(* Logix 5000 project; controller ecust2024 vendor 1 type 14 code 108 rev 30.11; software revision 30.00; part 2 of 2 *)
(* tags used below, declared in another part *)
   circle_count : DINT;
   circle_num1 : DINT;
   count11 : COUNTER;
   delay4 : TIMER;
   LED1 : LED_control;
   LED2 : LED_control;
   LED3 : LED_control;
   speed_dec : BOOL;
   speed_inc : BOOL;
   velocity : DINT;
   wait1 : TIMER;
   wait2 : TIMER;
   wait3 : TIMER;
   A : OneKey;
   anticlockwise : MOTION_INSTRUCTION;
   anticlockwise_order : BOOL;
   Axis_1 : AXIS_CIP_DRIVE;
   Change_speed : BOOL;
   changespeed : MOTION_INSTRUCTION;
   clockwise1 : MOTION_INSTRUCTION;
   clockwise_order : BOOL;
   count5 : COUNTER;
   count6 : COUNTER;
   Direction_Change3 : BOOL;
   Direction_Change4 : BOOL;
   Direction_change_state3 : BOOL;
   Holding_Cmd : BOOL;
   Light1 : BOOL;
   Light2 : BOOL;
   Light3 : BOOL;
   LT1 : BOOL;
   LT2 : BOOL;
   LT3 : BOOL;
   My_Equipment_Phase : PHASE;
   oneshot : DINT;
   Reset_Cmd : BOOL;
   Restart_Cmd : BOOL;
   S : DINT;
   Sensor1_cmd : BOOL;
   Sensor2_cmd : BOOL;
   setspeed : DINT;
   Start_Cmd : BOOL;
   Start_PB : BOOL;
   StartA : BOOL;
   Stop : MOTION_INSTRUCTION;
   Stop_Cmd : BOOL;
   Stop_PB : BOOL;
   Temp_CMX : REAL;
   temperature_speed : REAL;
   time1 : TIMER;
   time2 : TIMER;
   time4 : TIMER;
   ts : BOOL;
(* MainProgram, continued *)

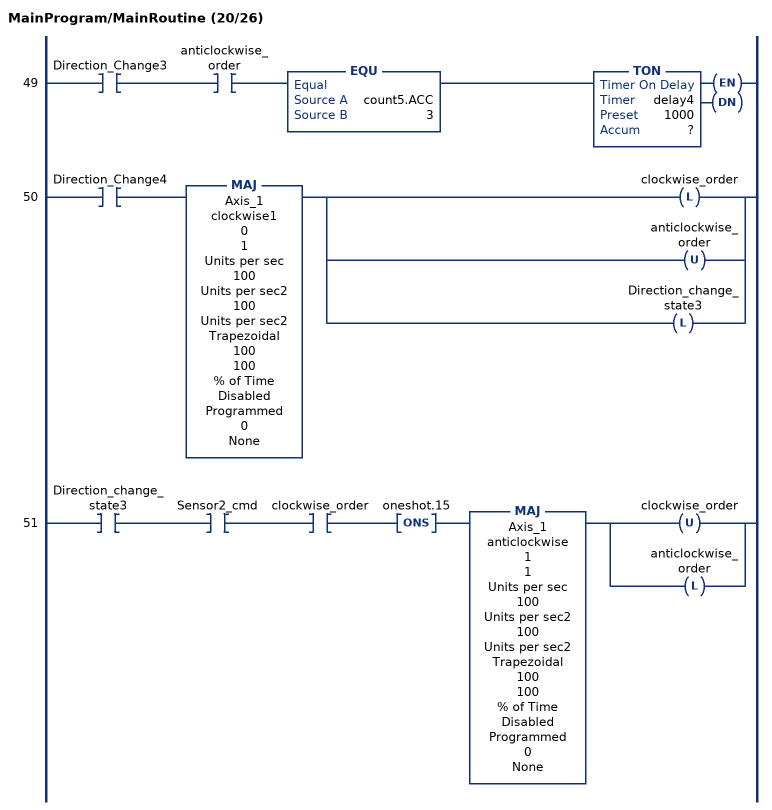
   [picture p25: MainProgram/MainRoutine rungs 49-51]
   49: XIC(Direction_Change3)XIC(anticlockwise_order)EQU(count5.ACC,3)TON(delay4,?,?);
   50: XIC(Direction_Change4)MAJ(Axis_1,clockwise1,0,1,Units per sec,100,Units per sec2,100,Units per sec2,Trapezoidal,100,100,% of Time,Disabled,Programmed,0,None)[OTL(clockwise_order) ,OTU(anticlockwise_order) ,OTL(Direction_change_state3) ];
   51: XIC(Direction_change_state3)XIC(Sensor2_cmd)XIC(clockwise_order)ONS(oneshot.15)MAJ(Axis_1,anticlockwise,1,1,Units per sec,100,Units per sec2,100,Units per sec2,Trapezoidal,100,100,% of Time,Disabled,Programmed,0,None)[OTU(clockwise_order) ,OTL(anticlockwise_order) ];
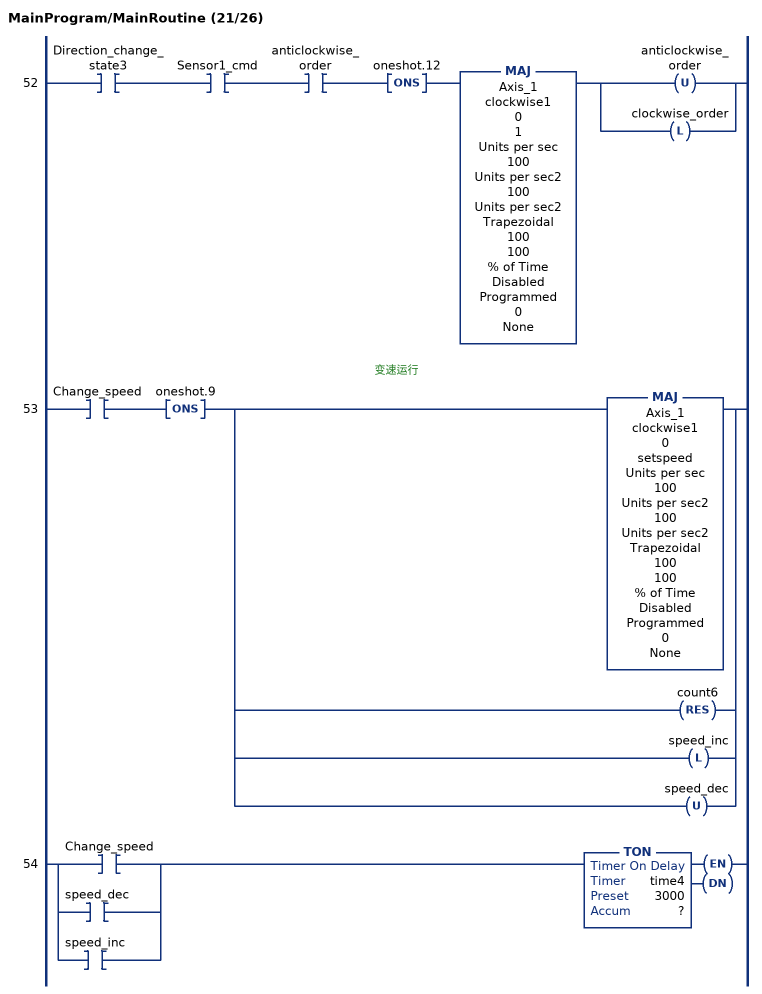
   52: XIC(Direction_change_state3)XIC(Sensor1_cmd)XIC(anticlockwise_order)ONS(oneshot.12)MAJ(Axis_1,clockwise1,0,1,Units per sec,100,Units per sec2,100,Units per sec2,Trapezoidal,100,100,% of Time,Disabled,Programmed,0,None)[OTU(anticlockwise_order) ,OTL(clockwise_order) ];
   // 变速运行
   53: XIC(Change_speed)ONS(oneshot.9)[MAJ(Axis_1,clockwise1,0,setspeed,Units per sec,100,Units per sec2,100,Units per sec2,Trapezoidal,100,100,% of Time,Disabled,Programmed,0,None) ,[RES(count6) ,OTL(speed_inc) ,OTU(speed_dec) ] ];
   54: [XIC(Change_speed) ,XIC(speed_dec) ,XIC(speed_inc) ]TON(time4,?,?);
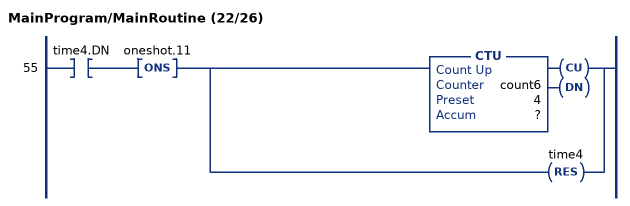
   55: XIC(time4.DN)ONS(oneshot.11)[CTU(count6,?,?) ,RES(time4) ];
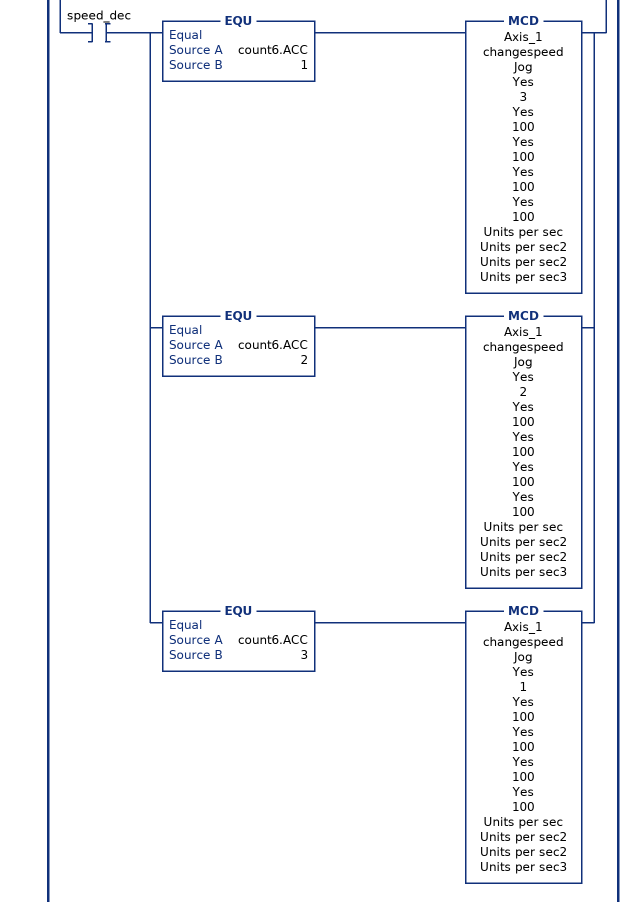
   56: [XIC(speed_inc) [EQU(count6.ACC,1) MCD(Axis_1,changespeed,Jog,Yes,1,Yes,100,Yes,100,Yes,100,Yes,100,Units per sec,Units per sec2,Units per sec2,Units per sec3) ,EQU(count6.ACC,2) MCD(Axis_1,changespeed,Jog,Yes,2,Yes,100,Yes,100,Yes,100,Yes,100,Units per sec,Units per sec2,Units per sec2,Units per sec3) ,EQU(count6.ACC,3) MCD(Axis_1,changespeed,Jog,Yes,3,Yes,100,Yes,100,Yes,100,Yes,100,Units per sec,Units per sec2,Units per sec2,Units per sec3) ] ,XIC(speed_dec) [EQU(count6.ACC,1) MCD(Axis_1,changespeed,Jog,Yes,3,Yes,100,Yes,100,Yes,100,Yes,100,Units per sec,Units per sec2,Units per sec2,Units per sec3) ,EQU(count6.ACC,2) MCD(Axis_1,changespeed,Jog,Yes,2,Yes,100,Yes,100,Yes,100,Yes,100,Units per sec,Units per sec2,Units per sec2,Units per sec3) ,EQU(count6.ACC,3) MCD(Axis_1,changespeed,Jog,Yes,1,Yes,100,Yes,100,Yes,100,Yes,100,Units per sec,Units per sec2,Units per sec2,Units per sec3) ] ];
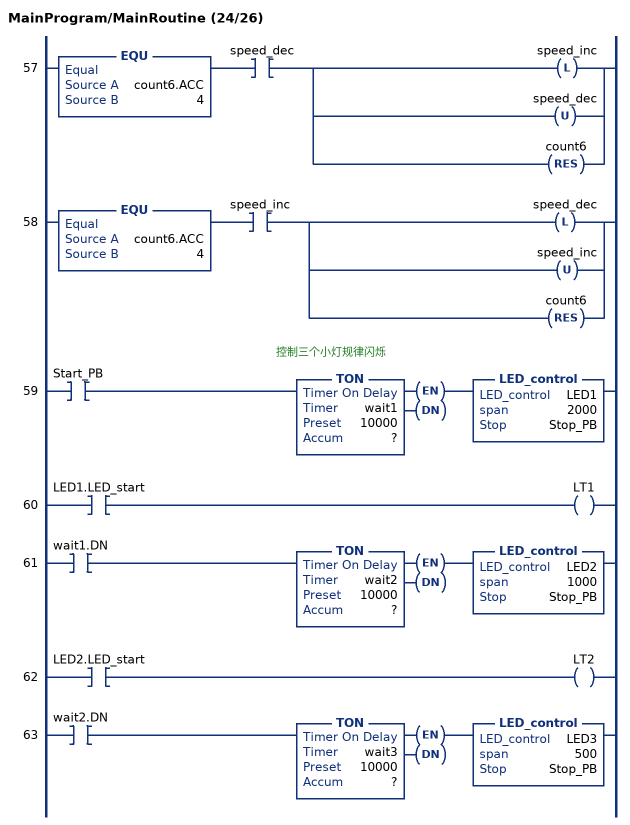
   57: EQU(count6.ACC,4)XIC(speed_dec)[OTL(speed_inc) ,OTU(speed_dec) ,RES(count6) ];
   58: EQU(count6.ACC,4)XIC(speed_inc)[OTL(speed_dec) ,OTU(speed_inc) ,RES(count6) ];
   // 控制三个小灯规律闪烁
   59: XIC(Start_PB)TON(wait1,?,?)LED_control(LED1,2000,Stop_PB);
   60: XIC(LED1.LED_start)OTE(LT1);
   61: XIC(wait1.DN)TON(wait2,?,?)LED_control(LED2,1000,Stop_PB);
   62: XIC(LED2.LED_start)OTE(LT2);
   63: XIC(wait2.DN)TON(wait3,?,?)LED_control(LED3,500,Stop_PB);
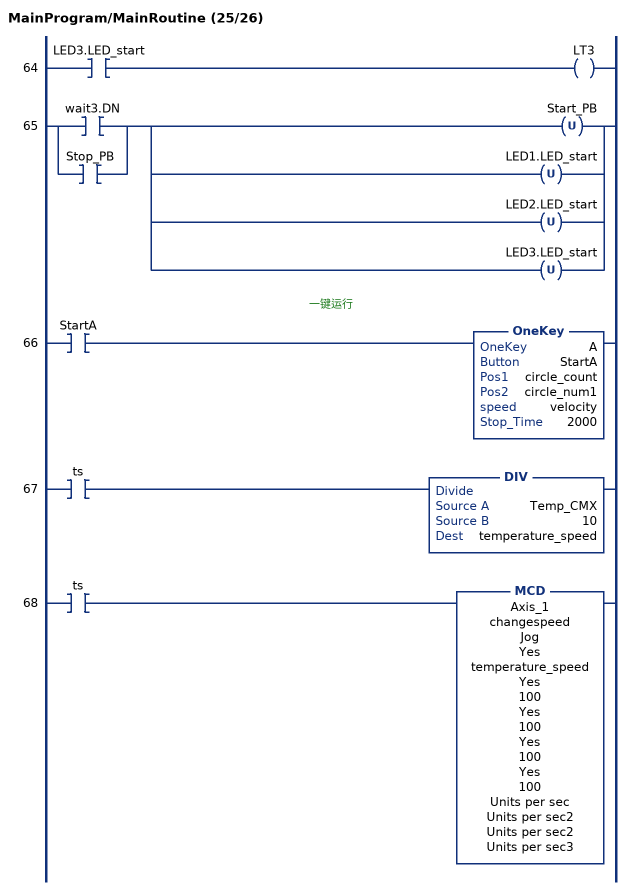
   64: XIC(LED3.LED_start)OTE(LT3);
   65: [XIC(wait3.DN) ,XIC(Stop_PB) ][OTU(Start_PB) ,OTU(LED1.LED_start) ,OTU(LED2.LED_start) ,OTU(LED3.LED_start) ];
   // 一键运行
   66: XIC(StartA)OneKey(A,StartA,circle_count,circle_num1,velocity,2000);
   67: XIC(ts)DIV(Temp_CMX,10,temperature_speed);
   68: XIC(ts)MCD(Axis_1,changespeed,Jog,Yes,temperature_speed,Yes,100,Yes,100,Yes,100,Yes,100,Units per sec,Units per sec2,Units per sec2,Units per sec3);
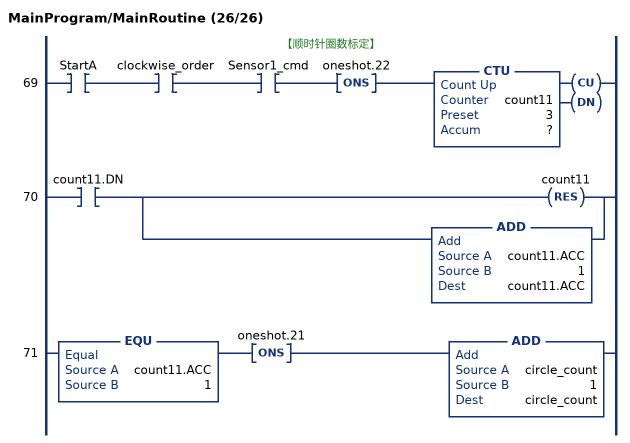
   // 【顺时针圈数标定】
   69: XIC(StartA)XIC(clockwise_order)XIC(Sensor1_cmd)ONS(oneshot.22)CTU(count11,?,?);
   70: XIC(count11.DN)[RES(count11) ,ADD(count11.ACC,1,count11.ACC) ];
   71: EQU(count11.ACC,1)ONS(oneshot.21)ADD(circle_count,1,circle_count);
END_ROUTINE
END_PROGRAM

PROGRAM My_Equipment_Phase
VAR
   FAL_M_CD : CONTROL := (LEN := 1);
   FAL_M_JOG : CONTROL := (LEN := 16);
   FAL_M_ServoOff : CONTROL := (LEN := 1);
   FAL_M_ServoOff_Stopping : CONTROL := (LEN := 1);
   FAL_M_ServoOn : CONTROL := (LEN := 1);
   FAL_M_Stop : CONTROL := (LEN := 1);
   FAL_M_Stop_Stopping : CONTROL := (LEN := 1);
   Holding_Result : DINT;
   M_CD_Axis_1 : MOTION_INSTRUCTION := (FLAGS := 570425344, DN := 1);
   M_Jog_Axis_1 : MOTION_INSTRUCTION := (FLAGS := 570425344, DN := 1);
   M_ServoOff_Axis_1 : MOTION_INSTRUCTION := (FLAGS := -2113929216, EN := 1, STATUS := 2, STATE := 1);
   M_ServoOff_Stopping : MOTION_INSTRUCTION := (FLAGS := -1577058304, EN := 1, DN := 1, STATUS := 2, STATE := 1);
   M_ServoOn_Axis_1 : MOTION_INSTRUCTION := (FLAGS := 570425344, DN := 1);
   M_Stop_Axis_1 : MOTION_INSTRUCTION := (FLAGS := 704643072, DN := 1, PC := 1);
   M_Stop_Stopping : MOTION_INSTRUCTION := (FLAGS := 704643072, DN := 1, PC := 1);
   Reset_Result : DINT;
   Restart_Result : DINT;
   Start_Result : DINT;
   Stop_Result : DINT;
   StoreONS : DINT;
   Timer1 : TIMER := (PRE := 5000);
   Timer1_temp : TIMER;
   Timer2 : TIMER := (PRE := 5000);
   Timer2_temp : TIMER;
   Timer3 : TIMER := (PRE := 3000);
   Timer3_temp : TIMER;
END_VAR

ROUTINE Holding   (* ladder *)
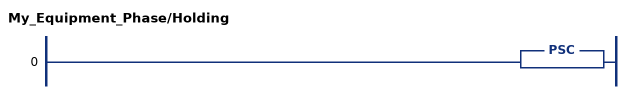
   0: PSC();
END_ROUTINE

ROUTINE Prestate   (* ladder *)
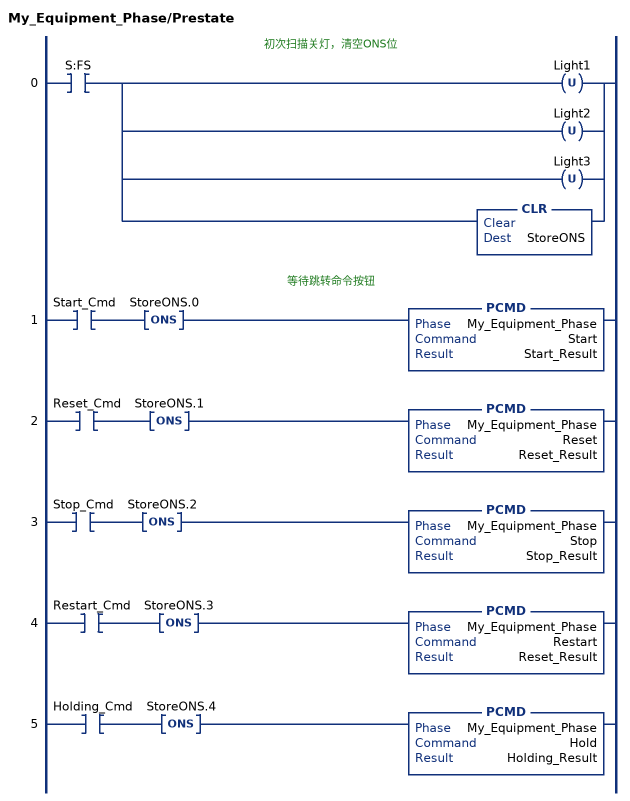
   // 初次扫描关灯，清空ONS位
   0: XIC(S:FS)[OTU(Light1) ,OTU(Light2) ,OTU(Light3) ,CLR(StoreONS) ];
   // 等待跳转命令按钮
   1: XIC(Start_Cmd)ONS(StoreONS.0)PCMD(My_Equipment_Phase,Start,Start_Result);
   2: XIC(Reset_Cmd)ONS(StoreONS.1)PCMD(My_Equipment_Phase,Reset,Reset_Result);
   3: XIC(Stop_Cmd)ONS(StoreONS.2)PCMD(My_Equipment_Phase,Stop,Stop_Result);
   4: XIC(Restart_Cmd)ONS(StoreONS.3)PCMD(My_Equipment_Phase,Restart,Reset_Result);
   5: XIC(Holding_Cmd)ONS(StoreONS.4)PCMD(My_Equipment_Phase,Hold,Holding_Result);
END_ROUTINE

ROUTINE Resetting   (* ladder *)
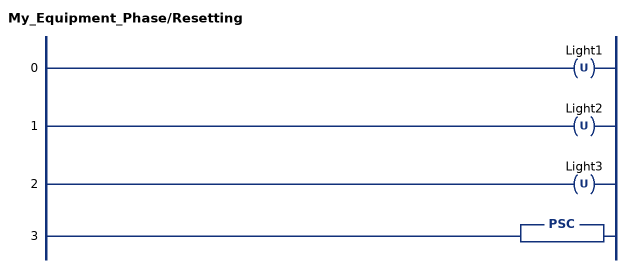
   0: OTU(Light1);
   1: OTU(Light2);
   2: OTU(Light3);
   3: PSC();
END_ROUTINE

ROUTINE Restarting   (* ladder *)
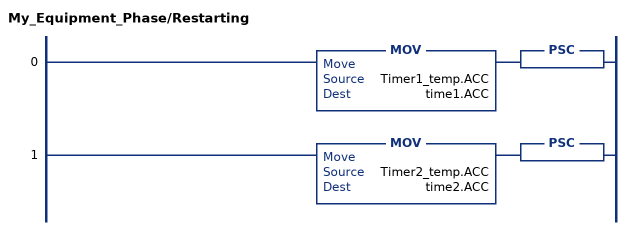
   0: MOV(Timer1_temp.ACC,time1.ACC)PSC();
   1: MOV(Timer2_temp.ACC,time2.ACC)PSC();
END_ROUTINE

ROUTINE Running   (* ladder *)
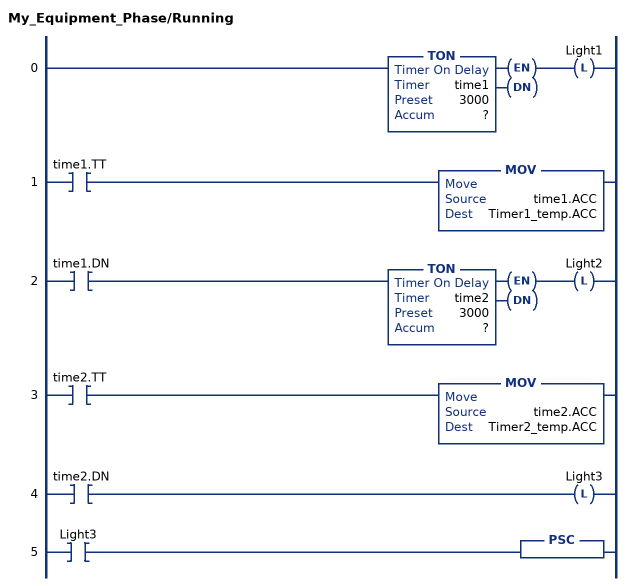
   0: TON(time1,?,?)OTL(Light1);
   1: XIC(time1.TT)MOV(time1.ACC,Timer1_temp.ACC);
   2: XIC(time1.DN)TON(time2,?,?)OTL(Light2);
   3: XIC(time2.TT)MOV(time2.ACC,Timer2_temp.ACC);
   4: XIC(time2.DN)OTL(Light3);
   5: XIC(Light3)PSC();
END_ROUTINE

ROUTINE Stopping   (* ladder *)
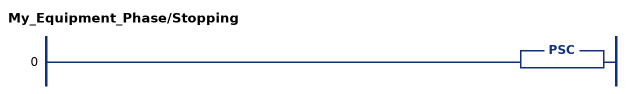
   0: PSC();
END_ROUTINE
END_PROGRAM
